# B&R Automation Studio project URTKtry3
Automation Studio 4.12.4.107 SP; technology packages: Acp10Arnc0 5.16.2

## Configuration Config1

CPU PC_any, AutomationRuntime C4.90, Build 4.1.2, Safety 0.0, Vc V4.72.2

### Task classes (Cpu.sw)
```
Cyclic#1:
  URTKPrg <- URTKFmu.URTKPrg.prg
NcDataObjects: AxInit <- URTKFmu.AxInit.dob, AcpParTab <- URTKFmu.AcpParTab.dob, acp10etxen <- acp10etxen.dob, gAxis01a <- gAxis01obj.gAxis01a.dob, gAxis01i <- gAxis01obj.gAxis01i.dob
Binaries: udbdef, FWRules, TCData, sysconf, Role, User, iomap, ashwd, asfw, arconfig, ashwac
Libraries: URTKLib, sys_lib, runtime, Coollb, Acp10man, Acp10par, NcGlobal, Acp10sdc, Acp10sim, Acp10_MC, brsystem, AsIoTime
```

### Hardware
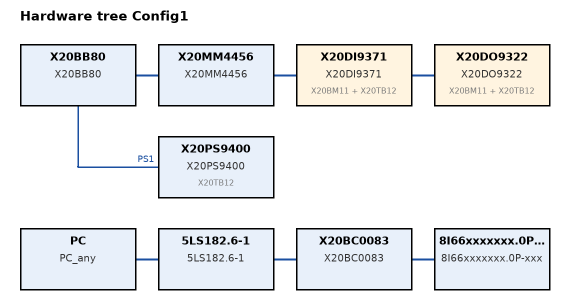
```
5LS182.6-1 : 5LS182.6-1 v1.5.0.0  [SL -> PC.SL1]
8I66xxxxxxx.0P-xxx : 8I66xxxxxxx.0P-xxx v2.5.1.0  [PLK1 -> X20BC0083.PLK2 (NodeNumber=2) [Cable Type=PowerlinkCable, Length=10, Version=1.0.0.3]]
  FunctionModel = MotionConfig
  UnitOfSetpoint = Rpm
PC : PC_any v1.1.1.0 (OrderNumber=PC)
  ConfigurationID = URTKtry3_Config1
  Cyclic1Tolerance = 0
  ActivateOpcUa = 1
  OpcUaInformationModels_PV_Version = 1
X20BB80 : X20BB80 v1.1.0.0
X20BC0083 : X20BC0083 v2.14.0.0  [PLK1 -> 5LS182.6-1.IF1 (NodeNumber=1) [Cable Type=PowerlinkCable, Length=10, Version=1.0.0.3]; PLK2 -> 8I66xxxxxxx.0P-xxx.PLK1 (NodeNumber=1) [Cable Type=PowerlinkCable, Length=10, Version=1.0.0.3]; SL -> X20BB80.SL1]
X20BM11 : X20BM11 v1.1.0.0  [X2X1 -> X20BM11a.X2X2]
X20BM11a : X20BM11 v1.1.0.0  [X2X1 -> X20MM4456.X2X2]
X20DI9371 : X20DI9371 v1.4.0.0  [SS1 -> X20TB12a.SS; SL -> X20BM11a.SL1]
X20DO9322 : X20DO9322 v1.5.0.0  [SS1 -> X20TB12b.SS; SL -> X20BM11.SL1]
X20MM4456 : X20MM4456 v1.5.0.0  [X2X1 -> X20BB80.IF1]
X20PS9400 : X20PS9400 v1.8.0.0  [SS1 -> X20TB12.SS; PS -> X20BB80.PS1]
X20TB12 : X20TB12 v1.0.0.0
X20TB12a : X20TB12 v1.0.0.0
X20TB12b : X20TB12 v1.0.0.0
```

### Acp10cfg.ncc - PC/Motion/Acp10cfg.ncc
```
NcConfiguration (Version=5.16.2, NcSwId=Acp10)
  ACP10CF1_typ:
    cnt_nettrc_rec_drive = 150
    bufsize_trace_upload = 1200
    tc_nc_man_task = Cyclic #1
    glob_pv_as_ncobject = Yes
    ncsys_dl_broadcast = Yes
    ncsys_dl_acp_reset = Yes
    safemc_log_err_to_ax = Yes
    network_init:
      ncsw_init_execute = Yes
      automatic_execute = No
      node_nr_warning = Yes
      net_err_before_ncact = Yes
    nettrc:
      enter_parsecrec = Yes
      enter_ncaction = Yes
      save_ring_startidx = No
    cam_prof_download:
      cam_dat_dl_parallel = No
      tc_cam_dl_parallel = Task class for NC Manager task
    sdc_if[0]:
      if_name = SDC_IF1
      mc_broadcast_size = 800
      mc_broadcast_extdat = No
```

### Acp10map1.ncm - PC/Motion/Acp10map1.ncm
```
NcMapping (NcSwId=ACP10, DisabledNodesAreHidden=False)
  NcObject Axis_X (ModuleAddress=SDC_IF1.ST1, InterfaceType=SDC, Type=ncAXIS, Channel=1, AcoposSimulation=Complete, InitParameter=AxInit, AcoposParameter=AcpParTab, Disabled=FALSE, ModuleDisabled=FALSE)
```

## Logical view

Binary libraries used (declarations not repeated): operator, runtime, astime, AsIecCon, sys_lib, Acp10man, Acp10par, NcGlobal, Acp10sdc, Acp10sim, Acp10_MC, brsystem, AsIoTime, URTKLib

### Global.var - Global variables
```iecst
VAR
	Axis_X : ACP10AXIS_typ;
	Axis_X_HW : SdcHwCfg_typ;
	Axis_X_DrvIf : SdcDrvIf16_typ;
	Axis_X_DiDoIf : SdcDiDoIf_typ;
	Axis_X_EncIf : SdcEncIf16_typ;
	Axis_Y : ACP10AXIS_typ;
	Axis_Y_HW : SdcHwCfg_typ;
	Axis_Y_DrvIf : SdcDrvIf16_typ;
	Axis_Y_DiDoIf : SdcDiDoIf_typ;
	Axis_Y_EncIf : SdcEncIf16_typ;
	Axis_Z : ACP10AXIS_typ;
	Axis_Z_HW : SdcHwCfg_typ;
	Axis_Z_DrvIf1 : SdcDrvIf16_typ;
	Axis_Z_DiDoIf : SdcDiDoIf_typ;
	Axis_Z_EncIf : SdcEncIf16_typ;
	gAxis01 : ACP10AXIS_typ;
END_VAR
```

### Package Logical/Libraries - Global libraries

### Library Logical/Libraries/Coollb (ANSIC)

#### Constants.var - Exported constants
```iecst
VAR CONSTANT
	d_t : REAL := 0.1;
END_VAR
```

### Program Logical/URTKFmu/URTKPrg (ANSIC)

#### Types.typ
```iecst
TYPE
	STATE_URTK :
		(
		ST_INIT,
		ST_READY,
		ST_HOME,
		ST_STOP,
		ST_MOVE
		);
END_TYPE
```

#### Variables.var
```iecst
VAR
	URTK1 : URTK := (0);
	URTKView_0 : URTKView := (0);
	urtk_out : URTK;
	sensorX1 : USINT;
	sensorX2 : USINT;
	sensorY1 : USINT;
	sensorY2 : USINT;
	sensorZ1 : USINT;
	sensorZ2 : USINT;
	statesURTK : STATE_URTK;
	fb_motor_z : FB_Motor;
	fb_motor_y : FB_Motor;
	fb_motor_x : FB_Motor;
	fb_controller : FB_Controller;
END_VAR
```

#### Cyclic.c
```c
#include <bur/plctypes.h>

#ifdef _DEFAULT_INCLUDES
#include <AsDefault.h>
#endif

void increase_counters(void);

void _CYCLIC ProgramCyclic(void)
{
	URTK(&URTK1);

	increase_counters();

	URTKView_0 .InstRef = URTK1.InstRef;

	URTKView(&URTKView_0 );

	urtk_out.internal_axisZ1 = URTK1.internal_axisZ1 + 252.315;
	urtk_out.internal_axisZ2 = URTK1.internal_axisZ2 + 336.641;
	urtk_out.internal_axisZ3 = URTK1.internal_axisZ3-50.1246;
	urtk_out.internal_axisY1 = URTK1.internal_axisY1 + 280.678;
	urtk_out.internal_axisY2 = URTK1.internal_axisY2 + 114.875;
	urtk_out.internal_axisY3 = URTK1.internal_axisY3 - 267.531;
	urtk_out.internal_Ground1 = URTK1.internal_Ground1 + 241.35;
	urtk_out.internal_Ground2 = URTK1.internal_Ground2 + 20.735;
	urtk_out.internal_Ground3 = URTK1.internal_Ground3 - 50.4717;
	urtk_out.internal_movementX1 = URTK1.internal_movementX1 + 253.027;
	urtk_out.internal_movementX2 = URTK1.internal_movementX2 + 38.0305;
	urtk_out.internal_movementX3 = URTK1.internal_movementX3 - 49.6654;
	urtk_out.internal_movementY1 = URTK1.internal_movementY1 + 281.057;
	urtk_out.internal_movementY2 = URTK1.internal_movementY2 + 116.335;
	urtk_out.internal_movementY3 = URTK1.internal_movementY3 - 48;
	urtk_out.internal_movementZ1 = URTK1.internal_movementZ1 + 252.937;
	urtk_out.internal_movementZ2 = URTK1.internal_movementZ2 + 117;
	urtk_out.internal_movementZ3 = URTK1.internal_movementZ3 - 48.6654;

	if (urtk_out.internal_movementX1 <= 80)
	{
		sensorX1 = 1;
	}

	if (urtk_out.internal_movementX1 >= 340)
	{
		sensorX2 = 1;
	}

	if (urtk_out.internal_movementX1 >= 80 && urtk_out.internal_movementX1 <= 340)
	{
		sensorX1 = 0;
		sensorX2 = 0;
	}

	if (urtk_out.internal_movementZ2 <= 130)
	{
		sensorY1 = 1;
	}

	if (urtk_out.internal_movementZ2 >= 390)
	{
		sensorY2 = 1;
	}

	if (urtk_out.internal_movementZ2 >= 130 && urtk_out.internal_movementZ2 <= 390)
	{
		sensorY1 = 0;
		sensorY2 = 0;
	}

	if (urtk_out.internal_axisY3 <= -255)
	{
		sensorZ1 = 1;
	}

	if (urtk_out.internal_axisY3 >= 10)
	{
		sensorZ2 = 1;
	}

	if (urtk_out.internal_axisY3 >= -255 && urtk_out.internal_axisY3 <= 10)
	{
		sensorZ1 = 0;
		sensorZ2 = 0;
	}

	Axis_X_EncIf.iActTime = (INT)	AsIOTimeCyclicStart();
	Axis_X_EncIf.iActPos = urtk_out.internal_movementX1*100;
	Axis_X_DiDoIf.iPosHwEnd = sensorX2;
	Axis_X_DiDoIf.iNegHwEnd = sensorX1;
	URTK1.Xinputvelocity = Axis_X_DrvIf.oSetPos * 1000.0 / 32767;

	/*

	if (urtk_out.internal_movementX1 <= 80)
	{
		sensorX1 = 1;
		if (URTK1.Xinputvelocity > 0)
			URTK1.Xinputvelocity = 0;
	}

	if (urtk_out.internal_movementX1 >= 340)
	{
		sensorX2 = 1;
		if (URTK1.Xinputvelocity < 0)
			URTK1.Xinputvelocity = 0;
	}

	if (urtk_out.internal_movementX1 >= 80 && urtk_out.internal_movementX1 <= 340)
	{
		sensorX1 = 0;
		sensorX2 = 0;
	}

	if (urtk_out.internal_movementZ2 <= 130)
	{
		sensorY1 = 1;
		if (URTK1.Zimputevelocity < 0)
			URTK1.Zimputevelocity = 0;
	}

	if (urtk_out.internal_movementZ2 >= 390)
	{
		sensorY2 = 1;
		if (URTK1.Zimputevelocity > 0)
			URTK1.Zimputevelocity = 0;
	}

	if (urtk_out.internal_movementZ2 >= 130 && urtk_out.internal_movementZ2 <= 390)
	{
		sensorY1 = 0;
		sensorY2 = 0;
	}

	if (urtk_out.internal_axisY3 <= -255)
	{
		sensorZ1 = 1;
		if (URTK1.Yimputvelocity < 0)
			URTK1.Yimputvelocity = 0;
	}

	if (urtk_out.internal_axisY3 >= 10)
	{
		sensorZ2 = 1;
		if (URTK1.Yimputvelocity > 0)
			URTK1.Yimputvelocity = 0;
	}

	if (urtk_out.internal_axisY3 >= -255 && urtk_out.internal_axisY3 <= 10)
	{
		sensorZ1 = 0;
		sensorZ2 = 0;
	}

	int max_speed = 1000;

	if (URTK1.Xinputvelocity>max_speed)
		URTK1.Xinputvelocity = max_speed;
	if (URTK1.Xinputvelocity<-max_speed)
		URTK1.Xinputvelocity = -max_speed;

	if (URTK1.Zimputevelocity>max_speed)
		URTK1.Zimputevelocity = max_speed;
	if (URTK1.Zimputevelocity<-max_speed)
		URTK1.Zimputevelocity = -max_speed;

	if (URTK1.Yimputvelocity>max_speed)
		URTK1.Yimputvelocity = max_speed;
	if (URTK1.Yimputvelocity<-max_speed)
		URTK1.Yimputvelocity = -max_speed;

	*/

}

void increase_counters(void)
{
	Axis_X_EncIf.iLifeCnt++;
	Axis_X_DiDoIf.iLifeCntDriveEnable++;
	Axis_X_DiDoIf.iLifeCntDriveReady++;
	Axis_X_DiDoIf.iLifeCntNegHwEnd++;
	Axis_X_DiDoIf.iLifeCntPosHwEnd++;
	Axis_X_DiDoIf.iLifeCntReference++;
	Axis_X_DrvIf.iLifeCnt++;
}
```

#### Init.c
```c
#include <bur/plctypes.h>

#ifdef _DEFAULT_INCLUDES
	#include <AsDefault.h>
#endif

void _INIT ProgramInit(void)
{
	urtk_out.internal_axisZ1 = 252.315;
	urtk_out.internal_axisZ2 = 336.641;
	urtk_out.internal_axisZ3 = -50.1246;
	urtk_out.internal_axisY1 = 280.678;
	urtk_out.internal_axisY2 = 114.875;
	urtk_out.internal_axisY3 = -267.531;
	urtk_out.internal_Ground1 = 241.35;
	urtk_out.internal_Ground2 = 20.735;
	urtk_out.internal_Ground3 = -50.4717;
	urtk_out.internal_movementX1 = 253.027;
	urtk_out.internal_movementX2 = 38.0305;
	urtk_out.internal_movementX3 = -49.6654;
	urtk_out.internal_movementY1 = 281.057;
	urtk_out.internal_movementY2 = 116.335;
	urtk_out.internal_movementY3 = -48;
	urtk_out.internal_movementZ1 = 252.937;
	urtk_out.internal_movementZ2 = 117;
	urtk_out.internal_movementZ3 = -48.6654;

	/*
	// Инициализация двигателей и регуляторов
	fb_motor_x.ke = 0;
	fb_motor_x.Tm = 0;

	fb_motor_y.ke = 0;
	fb_motor_y.Tm = 0;

	fb_motor_z.ke = 0;
	fb_motor_z.Tm = 0;

	fb_controller.k_i = 0;
	fb_controller.k_p = 0;
	fb_controller.max_abs_value = 24;
	*/
	//SDC Типы
	Axis_X_HW.EncIf1_Typ = ncSDC_ENC16;
	Axis_X_HW.DiDoIf_Typ = ncSDC_DIDO;
	Axis_X_HW.DrvIf_Typ = ncSDC_DRVSERVO16;

	//Устанавливаем имена переменных
	strcpy(Axis_X_HW.EncIf1_Name, "Axis_X_EncIf");
	strcpy(Axis_X_HW.DrvIf_Name, "Axis_X_DrvIf");
	strcpy(Axis_X_HW.DiDoIf_Name, "Axis_X_DiDoIf");

	//Устанавливаем входы готовности и нормальной работы
	Axis_X_EncIf.iEncOK = 1;
	Axis_X_DrvIf.iDrvOK = 1;
	Axis_X_DrvIf.iStatusEnable = 1;
	Axis_X_DiDoIf.iDriveReady = 1;

}
```

### Data object Logical/URTKFmu/AxInit (Ax)

#### AxInitAcp10.ax
```
InitParameter (Version=5.16.2, NcSwId=ACP10)
  ACP10AXIS_typ:
    dig_in:
      level:
        reference = ncACTIV_HI
        pos_hw_end = ncACTIV_HI
        neg_hw_end = ncACTIV_HI
        trigger1 = ncACTIV_HI
        trigger2 = ncACTIV_HI
    encoder_if:
      parameter:
        count_dir = ncSTANDARD
        scaling:
          load:
            units = 1
            rev_motor = 100
    limit:
      parameter:
        v_pos = 1200.0
        v_neg = 1200.0
        a1_pos = 6000.0
        a2_pos = 6000.0
        a1_neg = 6000.0
        a2_neg = 6000.0
        t_jolt = 0
        t_in_pos = 0
        pos_sw_end = 2000000000
        neg_sw_end = -2000000000
        ds_warning = 500
        ds_stop = 1000
        a_stop = 1.0e30
        dv_stop = 0
        dv_stop_mode = ncOFF
    controller:
      mode = ncPOSITION
      position:
        kv = 50
        tn = 0
        t_predict = 0.0004
        t_total = 0.0004
        p_max = 10000
        i_max = 0
      speed:
        kv = 2.0
        tn = 0
        t_filter = 0.0
        isq_filter1:
          type = ncOFF
          a0 = 0.0
          a1 = 0.0
          b0 = 0.0
          b1 = 0.0
          b2 = 0.0
          c0_par_id = 0
          c1_par_id = 0
        isq_filter2:
          type = ncOFF
          a0 = 0.0
          a1 = 0.0
          b0 = 0.0
          b1 = 0.0
          b2 = 0.0
          c0_par_id = 0
          c1_par_id = 0
        isq_filter3:
          type = ncOFF
          a0 = 0.0
          a1 = 0.0
          b0 = 0.0
          b1 = 0.0
          b2 = 0.0
          c0_par_id = 0
          c1_par_id = 0
      uf:
        type = ncLINEAR
        auto_config = ncMOTOR_PAR
        u0 = 0
        un = 0
        fn = 50.0
        k_f_slip = 0
      ff:
        mode = ncSTANDARD
        torque_load = 0.0
        torque_pos = 0.0
        torque_neg = 0.0
        kv_torque = 0.0
        inertia = 0.0
        t_filter_a = 0.0
      fb:
        mode = ncSTANDARD
        speed_mix_ratio = 0.0
        speed_kv = 2.0
      model:
        mass1:
          inertia = 0
          viscous_friction = 0
        mass2:
          inertia = 0
          viscous_friction = 0
          stiffness = 0
          damping = 0
    move:
      stop:
        parameter[0]:
          decel_ramp = ncA_LIMIT
          controller = ncON
        parameter[1]:
          decel_ramp = ncA_LIMIT
          controller = ncON
        parameter[2]:
          decel_ramp = ncA_LIMIT
          controller = ncON
        parameter[3]:
          decel_ramp = ncA_LIMIT
          controller = ncON
        quickstop:
          decel_ramp = ncA_LIMIT
          t_jolt = 0
        drive_error:
          decel_ramp = ncA_LIMIT
      homing:
        parameter:
          s = 0
          v_switch = 800.0
          v_trigger = 200.0
          a = 4800.0
          mode = ncEND_SWITCH
          edge_sw = ncNEGATIVE
          start_dir = ncPOSITIVE
          trigg_dir = ncNEGATIVE
          ref_pulse = ncOFF
          fix_dir = ncOFF
          tr_s_block = 0
          torque_lim = 0
          ds_block = 0
          ds_stop = 0
      basis:
        parameter:
          v_pos = 500.0
          v_neg = 500.0
          a1_pos = 3000.0
          a2_pos = 3000.0
          a1_neg = 3000.0
          a2_neg = 3000.0
    message:
      text:
        parameter:
          format = ncBREAK
          columns = 80
          data_modul
```

### Data object Logical/URTKFmu/AcpParTab (Apt)

#### AcpParTab.apt
```
AcoposParameterTable:
  Root Parameters:
    109 = 1 (Name=SCALE_ENCOD_INCR)  // Encoder1: Encoder scaling: increments per encoder revolution
    64201 = 1000 (Name=SERVO_V_MAX_OUTPUT, Unit=Units/s)  // Servo drive adjustment: Velocity at maximum output value
```

### Data object Logical/acp10etxen (Ett)

- acp10etxen.ett (not shown)

### Package Logical/gAxis01obj - gAxis01obj

### gAxis01i.ax
```
InitParameter (Version=5.16.2, NcSwId=Acp10)
  ACP10AXIS_typ:
    dig_in:
      level:
        reference = ncACTIV_HI
        pos_hw_end = ncACTIV_LO
        neg_hw_end = ncACTIV_LO
        trigger1 = ncACTIV_HI
        trigger2 = ncACTIV_LO + ncQUICKSTOP
    encoder_if:
      parameter:
        count_dir = ncSTANDARD
        scaling:
          load:
            units = 1000
            rev_motor = 1
    limit:
      parameter:
        v_pos = 10000
        v_neg = 10000
        a1_pos = 50000
        a2_pos = 50000
        a1_neg = 50000
        a2_neg = 50000
        t_jolt = 0
        t_in_pos = 0
        pos_sw_end = 2000000000
        neg_sw_end = -2000000000
        ds_warning = 500
        ds_stop = 1000
        a_stop = 1.0e30
        dv_stop = 0
        dv_stop_mode = ncOFF
    controller:
      mode = ncPOSITION
      position:
        kv = 50
        tn = 0
        t_predict = 0.0004
        t_total = 0.0004
        p_max = 1.0e30
        i_max = 0
      speed:
        kv = 2.0
        tn = 0
        t_filter = 0.0
        isq_filter1:
          type = ncOFF
          a0 = 0.0
          a1 = 0.0
          b0 = 0.0
          b1 = 0.0
          b2 = 0.0
          c0_par_id = 0
          c1_par_id = 0
        isq_filter2:
          type = ncOFF
          a0 = 0.0
          a1 = 0.0
          b0 = 0.0
          b1 = 0.0
          b2 = 0.0
          c0_par_id = 0
          c1_par_id = 0
        isq_filter3:
          type = ncOFF
          a0 = 0.0
          a1 = 0.0
          b0 = 0.0
          b1 = 0.0
          b2 = 0.0
          c0_par_id = 0
          c1_par_id = 0
      uf:
        type = ncLINEAR + ncCORRECTION
        auto_config = ncMOTOR_PAR
        u0 = 0
        un = 0
        fn = 50.0
        k_f_slip = 0
      ff:
        mode = ncSTANDARD
        torque_load = 0.0
        torque_pos = 0.0
        torque_neg = 0.0
        kv_torque = 0.0
        inertia = 0.0
        t_filter_a = 0.0
      fb:
        mode = ncSTANDARD
        speed_mix_ratio = 0.0
        speed_kv = 2.0
      model:
        mass1:
          inertia = 0
          viscous_friction = 0
        mass2:
          inertia = 0
          viscous_friction = 0
          stiffness = 0
          damping = 0
    move:
      stop:
        parameter[0]:
          decel_ramp = ncA_LIMIT
          controller = ncON
        parameter[1]:
          decel_ramp = ncA_LIMIT
          controller = ncON
        parameter[2]:
          decel_ramp = ncA_LIMIT
          controller = ncON
        parameter[3]:
          decel_ramp = ncA_LIMIT
          controller = ncON
        quickstop:
          decel_ramp = ncA_LIMIT
          t_jolt = 0
        drive_error:
          decel_ramp = ncA_LIMIT
      homing:
        parameter:
          s = 0
          v_switch = 5000
          v_trigger = 500
          a = 50000
          mode = ncDIRECT
          edge_sw = ncPOSITIVE
          start_dir = ncPOSITIVE
          trigg_dir = ncPOSITIVE
          ref_pulse = ncOFF
          fix_dir = ncOFF
          tr_s_block = 0
          torque_lim = 0
          ds_block = 0
          ds_stop = 0
      basis:
        parameter:
          v_pos = 5000
          v_neg = 5000
          a1_pos = 50000
          a2_pos = 50000
          a1_neg = 50000
          a2_neg = 50000
    message:
      text:
        parameter:
          format = ncBREAK
          columns = 80
          data_modul = acp10etxen
```

Listed in the project but not available here: Logical/Global.typ, Logical/Libraries/Coollb/Types.typ, Logical/Libraries/Coollb/Coollb.fun, Logical/Libraries/Coollb/FB_motor.c, Logical/Libraries/Coollb/FB_Integrator.c, Logical/Libraries/Coollb/FB_Controller.c
